FUNCTION F_RectIntersectRect : BOOL
VAR_INPUT
	stRect1 : FB_Rectangle;
	stRect2 : FB_Rectangle;
END_VAR
VAR
END_VAR

//schneidet Rechteck1 Rechteck2?
F_RectIntersectRect := TRUE;
IF stRect1.X1 > stRect2.X2 OR stRect2.X1 > stRect1.X2 THEN
	F_RectIntersectRect := FALSE;
END_IF

IF stRect1.Y1 > stRect2.Y2 OR stRect2.Y1 > stRect1.Y2 THEN
	F_RectIntersectRect := FALSE;
END_IF

END_FUNCTION

(* stored: Version 1.1.0.1, ProductVersion 3.1.4022.18
   POU F_RectIntersectRect: Id {11e4e757-f481-41ae-8f93-23890945945a}, SpecialFunc None *)
